// TIA Portal V15.1 export
// export: Created 2024-06-21T08:41:01.5475302Z, ExportSetting WithDefaults, DisplayName Totally Integrated Automation Portal, DisplayVersion V15.1 Update 5, DisplayName TIA Portal Openness, DisplayVersion V15.1 Update 5, DisplayName SINAMICS Startdrive Advanced, DisplayVersion V15.1, DisplayName G130, G150, S120, S150, SINAMICS MV, S210, DisplayVersion V15.1, DisplayName G110M, G120, G120C, G120D, G120P, DisplayVersion V15.1, DisplayName STEP 7 Professional, DisplayVersion V15.1 Update 5, DisplayName STEP 7 Safety, DisplayVersion V15.1, DisplayName WinCC Professional, DisplayVersion V15.1 Update 5, DisplayName SIMATIC Visualization Architect, DisplayVersion V15.1
FUNCTION_BLOCK "LPassivate"   // FB1420, FBD
TITLE = LPassivate
{ S7_Optimized_Access := 'FALSE' }
AUTHOR : VCC
FAMILY : AlarmHnd
NAME : Passivat
VERSION : 0.1
// ================================================================================
// This module is used everywhere passivation of a slot shall generate an alarm.
// The alarm can be True only when the input Enable Alarm is also True.
// When the condition to generate the alarm is not fullfilled, a boolean output is 
// available to inform the upper level that the alarm can be reset.
// The alarm is reset by means of the AlarmResetPB signal.
// ================================================================================
// stored: AutoNumber false, IsIECCheckEnabled false, SetENOAutomatically False, UDAEnableTagReadback false
   VAR_INPUT
      I_SafetyCard_PASS_OUT { ExternalAccessible := 'False'; ExternalVisible := 'False'; ExternalWritable := 'False'} : Bool;   // Automatically generated DB from F-Modul (F-Peripherie DB)
      I_SafetyCard_ACK_REQ { ExternalAccessible := 'False'; ExternalVisible := 'False'; ExternalWritable := 'False'} : Bool;   // Automatically generated DB from F-Modul (F-Peripherie DB)
      I_SafetyCard_DIAG { ExternalAccessible := 'False'; ExternalVisible := 'False'; ExternalWritable := 'False'} : Byte;   // Automatically generated DB from F-Modul (F-Peripherie DB)
      I_SafetyCardHWSub { ExternalAccessible := 'False'; ExternalVisible := 'False'; ExternalWritable := 'False'} : HW_SUBMODULE;   // Safety I/O connection hardware
      I_AlarmClass { ExternalAccessible := 'False'; ExternalVisible := 'False'; ExternalWritable := 'False'} : Char;   // Alarm class -> A - B - C - D or E
      I_EnableAlarm { ExternalAccessible := 'False'; ExternalVisible := 'False'; ExternalWritable := 'False'} : Bool := TRUE;   // Enable alarm from upper level
      I_AlarmResetPB { ExternalAccessible := 'False'; ExternalVisible := 'False'; ExternalWritable := 'False'} : Bool;   // Alarm reset pushbutton is activated
      C_OutputCard { ExternalAccessible := 'False'; ExternalVisible := 'False'; ExternalWritable := 'False'} : Bool;   // 1 = The safety card is an output card
   END_VAR
   VAR_OUTPUT
      O_PassivateAlm { ExternalAccessible := 'False'; ExternalVisible := 'False'; ExternalWritable := 'False'} : Bool;   // Alarm
      O_AlarmABCondition { ExternalAccessible := 'False'; ExternalVisible := 'False'; ExternalWritable := 'False'} : Bool;   // Alarm AB condition
      H_IAnim { ExternalAccessible := 'False'; ExternalVisible := 'False'; ExternalWritable := 'False'} : Word;   // Icon animation
   END_VAR
   VAR DB_SPECIFIC
      H_Out : Struct   // HMI
         Anim : Word;   // HMI Animation of the object
         DBnr : Int;   // HMI Animation DB number
      END_STRUCT;
      Alarm { ExternalAccessible := 'False'; ExternalVisible := 'False'; ExternalWritable := 'False'} : Bool;   // Alarm
      AlarmClass_A { ExternalAccessible := 'False'; ExternalVisible := 'False'; ExternalWritable := 'False'} : Bool;   // The alarm is from alarm class A
      AlarmClass_B { ExternalAccessible := 'False'; ExternalVisible := 'False'; ExternalWritable := 'False'} : Bool;   // The alarm is from alarm class B
      AlarmClass_C { ExternalAccessible := 'False'; ExternalVisible := 'False'; ExternalWritable := 'False'} : Bool;   // The alarm is from alarm class C
      AlarmClass_D { ExternalAccessible := 'False'; ExternalVisible := 'False'; ExternalWritable := 'False'} : Bool;   // The alarm is from alarm class D
      AlarmCond { ExternalAccessible := 'False'; ExternalVisible := 'False'; ExternalWritable := 'False'} : Bool;   // Alarm condition
      QbadCh0 { ExternalAccessible := 'False'; ExternalVisible := 'False'; ExternalWritable := 'False'} : Bool;   // Passivation first Channel
      QbadCh1 { ExternalAccessible := 'False'; ExternalVisible := 'False'; ExternalWritable := 'False'} : Bool;   // Passivation second Channel
      QbadCh2 { ExternalAccessible := 'False'; ExternalVisible := 'False'; ExternalWritable := 'False'} : Bool;   // Passivation third Channel
      QbadCh3 { ExternalAccessible := 'False'; ExternalVisible := 'False'; ExternalWritable := 'False'} : Bool;   // Passivation fourth Channel
      Ack_Req { ExternalAccessible := 'False'; ExternalVisible := 'False'; ExternalWritable := 'False'} : Bool;   // Acknowledgement request
      Pass_Out { ExternalAccessible := 'False'; ExternalVisible := 'False'; ExternalWritable := 'False'} : Bool;   // Slot is passivated
      Timeout_F_I_O { ExternalAccessible := 'False'; ExternalVisible := 'False'; ExternalWritable := 'False'} : Bool;   // Timeout detected by F-I/O
      ChannelFault_F_I_O { ExternalAccessible := 'False'; ExternalVisible := 'False'; ExternalWritable := 'False'} : Bool;   // F-I/O fault or channel fault detected by F-I/O
      CRCSeqError_F_I_O { ExternalAccessible := 'False'; ExternalVisible := 'False'; ExternalWritable := 'False'} : Bool;   // CRC error or sequence number error detected by F-I/O
      Timeout_F_Sys { ExternalAccessible := 'False'; ExternalVisible := 'False'; ExternalWritable := 'False'} : Bool;   // Timeout detected by F-System
      SeqError_F_Sys { ExternalAccessible := 'False'; ExternalVisible := 'False'; ExternalWritable := 'False'} : Bool;   // Sequence number error detected by F-system
      CRCError_F_Sys { ExternalAccessible := 'False'; ExternalVisible := 'False'; ExternalWritable := 'False'} : Bool;   // CRC error detected by F-system
      RetValueData { ExternalAccessible := 'False'; ExternalVisible := 'False'; ExternalWritable := 'False'} : Int;   // Status variable (SFC14)
      DBnr { ExternalAccessible := 'False'; ExternalVisible := 'False'; ExternalWritable := 'False'} : Int;   // HMI DB number
   END_VAR
   VAR_TEMP
      T_DataFromSafetyCard : Struct   // Temp structure : receive data's from Safety Card
         Byte0_Bit0_QBadCh0 : Bool;
         Byte0_Bit1_QBadCh1 : Bool;
         Byte0_Bit2_QBadCh2 : Bool;
         Byte0_Bit3_QBadCh3 : Bool;
         Byte0_Bit4_Spare : Bool;
         Byte0_Bit5_Spare : Bool;
         Byte0_Bit6_Spare : Bool;
         Byte0_Bit7_Spare : Bool;
         Byte1_Bit0_QBadCh0 : Bool;
         Byte1_Bit1_QBadCh1 : Bool;
         Byte1_Bit2_QBadCh2 : Bool;
         Byte1_Bit3_QBadCh3 : Bool;
         Byte1_Bit4_Spare : Bool;
         Byte1_Bit5_Spare : Bool;
         Byte1_Bit6_Spare : Bool;
         Byte1_Bit7_Spare : Bool;
         Byte2_bit0_Spare : Bool;
         Byte2_bit1_Spare : Bool;
         Byte2_bit2_Spare : Bool;
         Byte2_bit3_Spare : Bool;
         Byte2_bit4_Spare : Bool;
         Byte2_bit5_Spare : Bool;
         Byte2_bit6_Spare : Bool;
         Byte2_bit7_Spare : Bool;
         Byte3_Bit0_Spare : Bool;
         Byte3_Bit1_Spare : Bool;
         Byte3_Bit2_Spare : Bool;
         Byte3_Bit3_Spare : Bool;
         Byte3_Bit4_Spare : Bool;
         Byte3_Bit5_Spare : Bool;
         Byte3_Bit6_Spare : Bool;
         Byte3_Bit7_Spare : Bool;
         Byte4_bit0_Spare : Bool;
         Byte4_bit1_Spare : Bool;
         Byte4_bit2_Spare : Bool;
         Byte4_bit3_Spare : Bool;
         Byte4_bit4_Spare : Bool;
         Byte4_bit5_Spare : Bool;
         Byte4_bit6_Spare : Bool;
         Byte4_bit7_Spare : Bool;
         Byte5_bit0_Spare : Bool;
         Byte5_bit1_Spare : Bool;
         Byte5_bit2_Spare : Bool;
         Byte5_bit3_Spare : Bool;
         Byte5_bit4_Spare : Bool;
         Byte5_bit5_Spare : Bool;
         Byte5_bit6_Spare : Bool;
         Byte5_bit7_Spare : Bool;
      END_STRUCT;
   END_VAR
BEGIN

NETWORK
TITLE = **** 1 - Inputs **** DB number
// DB number
      L     DINO;
      T     #DBnr;

NETWORK
TITLE = **** 1 - Inputs **** Alarm class
// Alarm class
// Alarm class = D
      L     #I_AlarmClass;
      L     'D';
      ==I;
      =     #AlarmClass_D;

// Alarm class = C
      L     #I_AlarmClass;
      L     'C';
      ==I;
      =     #AlarmClass_C;

// Alarm class = B
      L     #I_AlarmClass;
      L     'B';
      ==I;
      =     #AlarmClass_B;

// Alarm class = A
      AN    #AlarmClass_B;
      AN    #AlarmClass_C;
      AN    #AlarmClass_D;
      =     #AlarmClass_A;


REGION Network 3: **** 1 - Inputs **** Safety I/O connection hardware
   // Safety I/O connection hardware
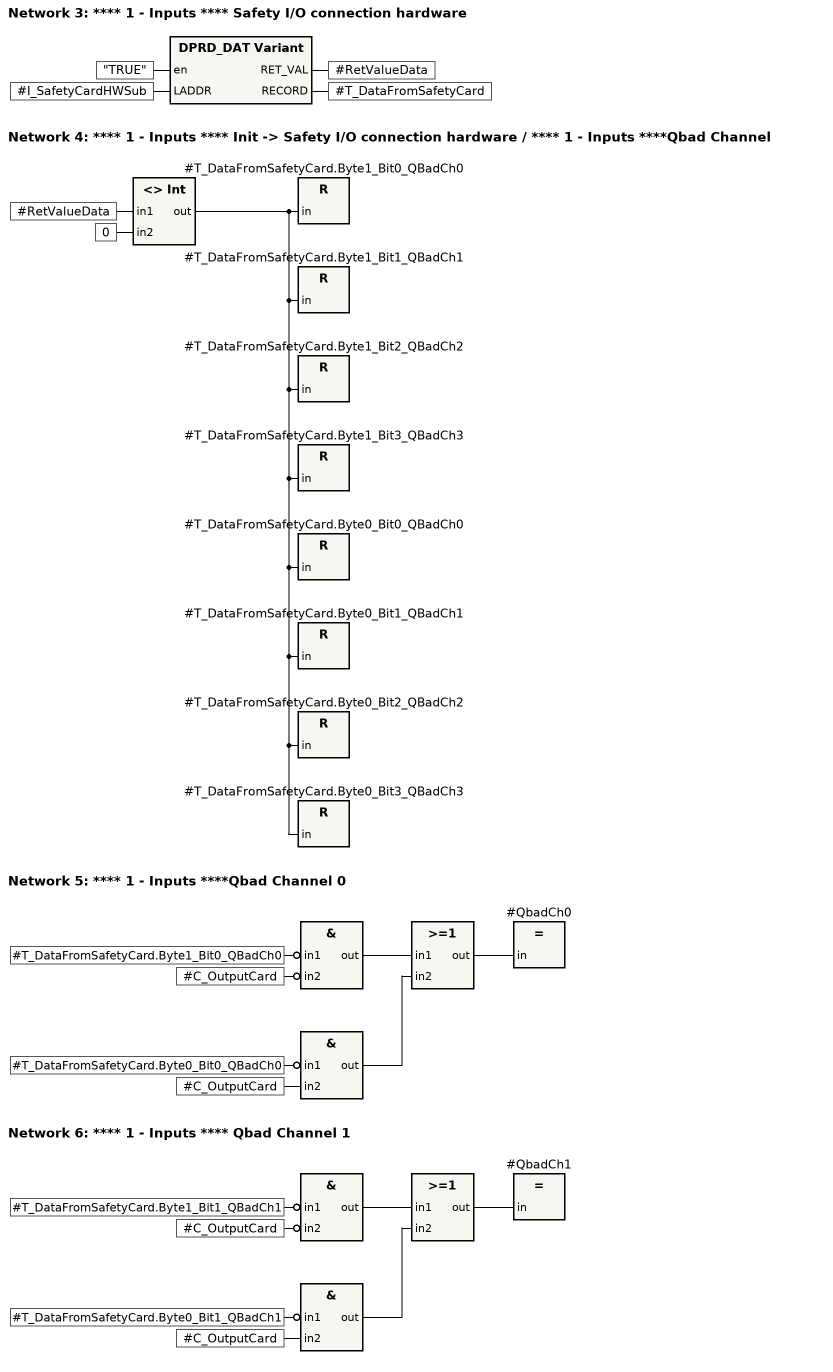
   IF "TRUE" THEN
       #RetValueData := DPRD_DAT(LADDR := #I_SafetyCardHWSub, RECORD => #T_DataFromSafetyCard);
   END_IF;
END_REGION

REGION Network 4: **** 1 - Inputs **** Init -> Safety I/O connection hardware / **** 1 - Inputs ****Qbad Channel
   // Init -> Safety I/O connection hardware
   IF #RetValueData <> 0 THEN
       #T_DataFromSafetyCard.Byte1_Bit0_QBadCh0 := FALSE;
       #T_DataFromSafetyCard.Byte1_Bit1_QBadCh1 := FALSE;
       #T_DataFromSafetyCard.Byte1_Bit2_QBadCh2 := FALSE;
       #T_DataFromSafetyCard.Byte1_Bit3_QBadCh3 := FALSE;
       #T_DataFromSafetyCard.Byte0_Bit0_QBadCh0 := FALSE;
       #T_DataFromSafetyCard.Byte0_Bit1_QBadCh1 := FALSE;
       #T_DataFromSafetyCard.Byte0_Bit2_QBadCh2 := FALSE;
       #T_DataFromSafetyCard.Byte0_Bit3_QBadCh3 := FALSE;
   END_IF;
END_REGION

REGION Network 5: **** 1 - Inputs ****Qbad Channel 0
   // Qbad Channel 0
   #QbadCh0 := (NOT #T_DataFromSafetyCard.Byte1_Bit0_QBadCh0 AND NOT #C_OutputCard) OR (NOT #T_DataFromSafetyCard.Byte0_Bit0_QBadCh0 AND #C_OutputCard);
END_REGION

REGION Network 6: **** 1 - Inputs **** Qbad Channel 1
   // Qbad Channel 1
   #QbadCh1 := (NOT #T_DataFromSafetyCard.Byte1_Bit1_QBadCh1 AND NOT #C_OutputCard) OR (NOT #T_DataFromSafetyCard.Byte0_Bit1_QBadCh1 AND #C_OutputCard);
END_REGION

REGION Network 7: **** 1 - Inputs **** Qbad Channel 2
   // Qbad Channel 2
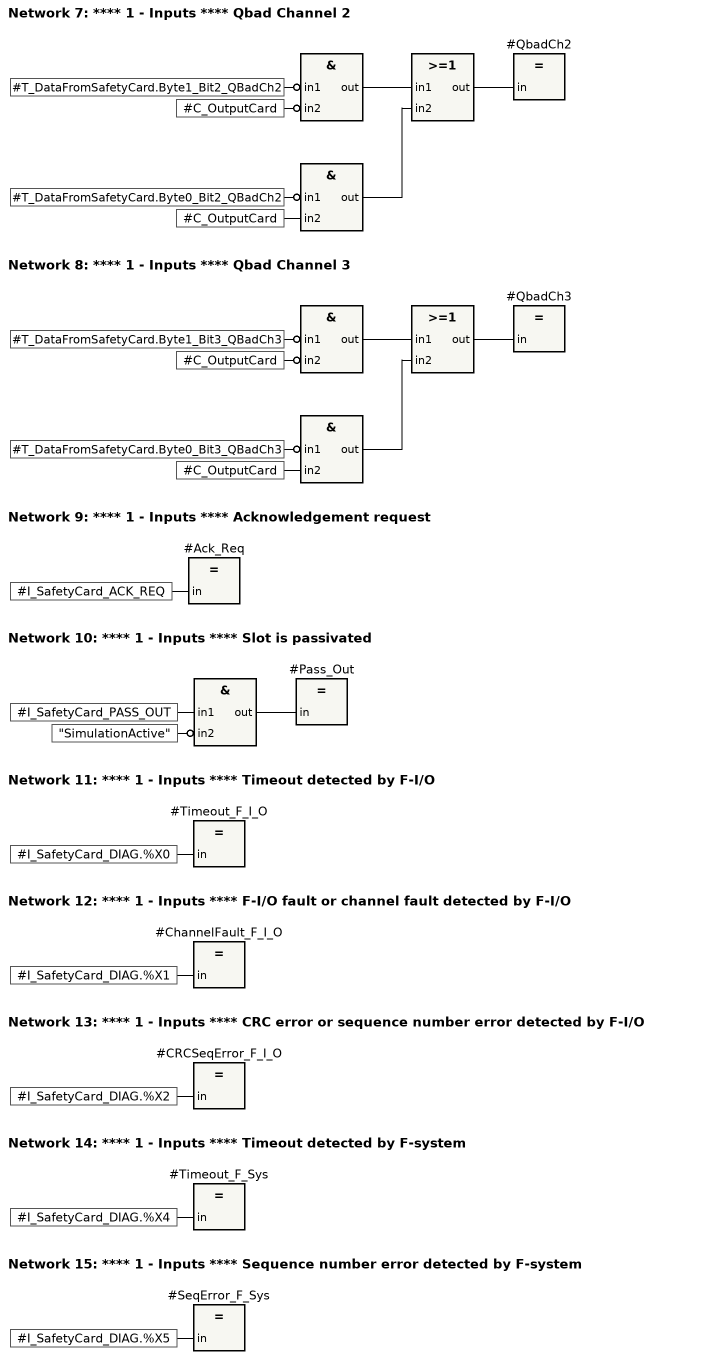
   #QbadCh2 := (NOT #T_DataFromSafetyCard.Byte1_Bit2_QBadCh2 AND NOT #C_OutputCard) OR (NOT #T_DataFromSafetyCard.Byte0_Bit2_QBadCh2 AND #C_OutputCard);
END_REGION

REGION Network 8: **** 1 - Inputs **** Qbad Channel 3
   // Qbad Channel 3
   #QbadCh3 := (NOT #T_DataFromSafetyCard.Byte1_Bit3_QBadCh3 AND NOT #C_OutputCard) OR (NOT #T_DataFromSafetyCard.Byte0_Bit3_QBadCh3 AND #C_OutputCard);
END_REGION

REGION Network 9: **** 1 - Inputs **** Acknowledgement request
   // Acknowledgement request
   #Ack_Req := #I_SafetyCard_ACK_REQ;
END_REGION

REGION Network 10: **** 1 - Inputs **** Slot is passivated
   // Slot is passivated
   #Pass_Out := #I_SafetyCard_PASS_OUT AND NOT "SimulationActive";
END_REGION

REGION Network 11: **** 1 - Inputs **** Timeout detected by F-I/O
   // Timeout detected by F-I/O
   #Timeout_F_I_O := #I_SafetyCard_DIAG.%X0;
END_REGION

REGION Network 12: **** 1 - Inputs **** F-I/O fault or channel fault detected by F-I/O
   // F-I/O fault or channel fault detected by F-I/O
   #ChannelFault_F_I_O := #I_SafetyCard_DIAG.%X1;
END_REGION

REGION Network 13: **** 1 - Inputs **** CRC error or sequence number error detected by F-I/O
   // CRC error or sequence number error detected by F-I/O
   #CRCSeqError_F_I_O := #I_SafetyCard_DIAG.%X2;
END_REGION

REGION Network 14: **** 1 - Inputs **** Timeout detected by F-system
   // Timeout detected by F-system
   #Timeout_F_Sys := #I_SafetyCard_DIAG.%X4;
END_REGION

REGION Network 15: **** 1 - Inputs **** Sequence number error detected by F-system
   // Sequence number error detected by F-system
   #SeqError_F_Sys := #I_SafetyCard_DIAG.%X5;
END_REGION

REGION Network 16: **** 1 - Inputs **** CRC error detected by F-system
   // CRC error detected by F-system
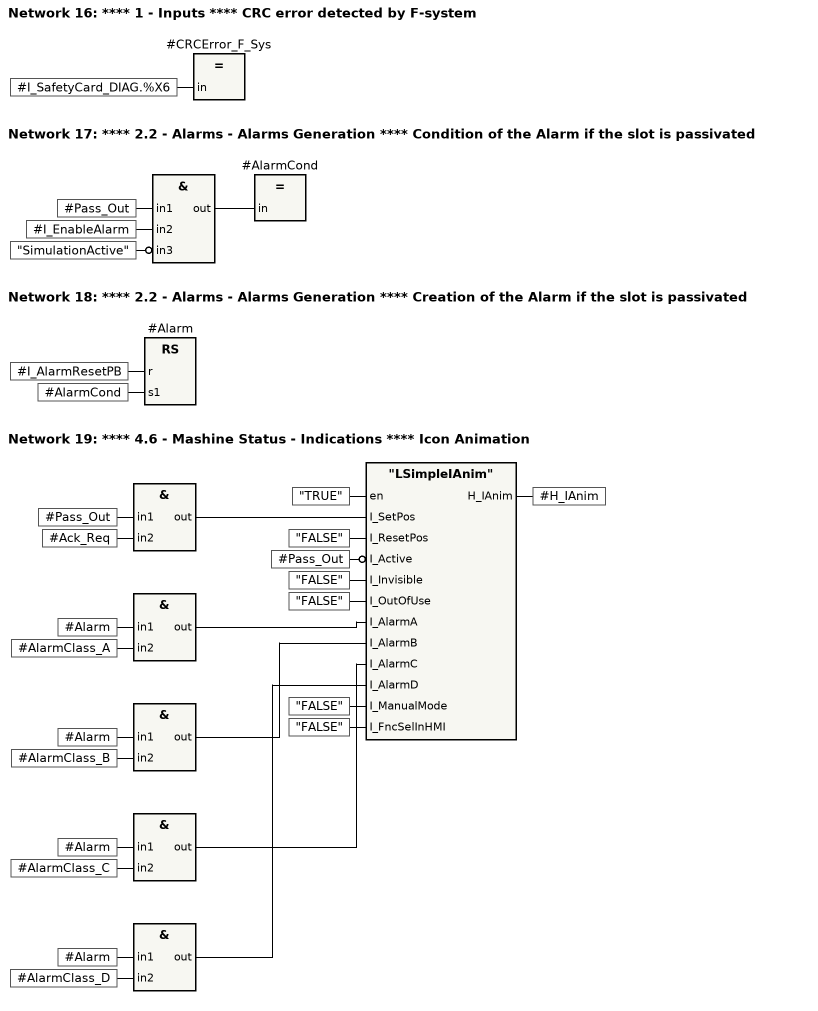
   #CRCError_F_Sys := #I_SafetyCard_DIAG.%X6;
END_REGION

REGION Network 17: **** 2.2 - Alarms - Alarms Generation **** Condition of the Alarm if the slot is passivated
   // Condition of the Alarm if the slot is passivated
   #AlarmCond := #Pass_Out AND #I_EnableAlarm AND NOT "SimulationActive";
END_REGION

REGION Network 18: **** 2.2 - Alarms - Alarms Generation **** Creation of the Alarm if the slot is passivated
   // Creation of the Alarm if the slot is passivated
   IF #I_AlarmResetPB THEN
       #Alarm := FALSE;   // RS flip-flop
   END_IF;
   IF #AlarmCond THEN #Alarm := TRUE; END_IF;
END_REGION

REGION Network 19: **** 4.6 - Mashine Status - Indications **** Icon Animation
   // Icon Animation
   IF "TRUE" THEN
       "LSimpleIAnim"(I_SetPos := #Pass_Out AND #Ack_Req,
                      I_ResetPos := "FALSE",
                      I_Active := NOT #Pass_Out,
                      I_Invisible := "FALSE",
                      I_OutOfUse := "FALSE",
                      I_AlarmA := #Alarm AND #AlarmClass_A,
                      I_AlarmB := #Alarm AND #AlarmClass_B,
                      I_AlarmC := #Alarm AND #AlarmClass_C,
                      I_AlarmD := #Alarm AND #AlarmClass_D,
                      I_ManualMode := "FALSE",
                      I_FncSelInHMI := "FALSE",
                      H_IAnim => #H_IAnim);
   END_IF;
END_REGION

REGION Network 20: **** 4.6 - Mashine Status - Indications **** Animation
   // Animation
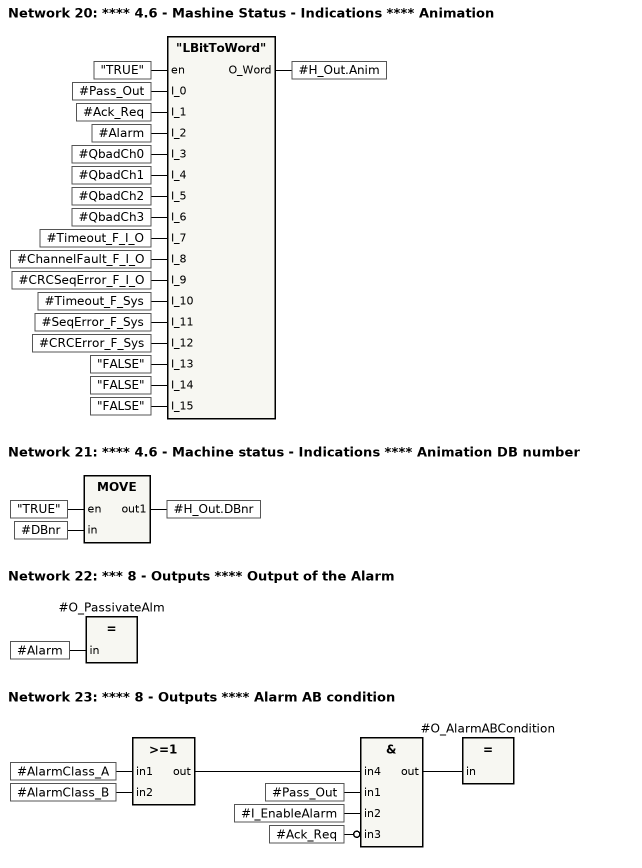
   IF "TRUE" THEN
       "LBitToWord"(I_0 := #Pass_Out,
                    I_1 := #Ack_Req,
                    I_2 := #Alarm,
                    I_3 := #QbadCh0,
                    I_4 := #QbadCh1,
                    I_5 := #QbadCh2,
                    I_6 := #QbadCh3,
                    I_7 := #Timeout_F_I_O,
                    I_8 := #ChannelFault_F_I_O,
                    I_9 := #CRCSeqError_F_I_O,
                    I_10 := #Timeout_F_Sys,
                    I_11 := #SeqError_F_Sys,
                    I_12 := #CRCError_F_Sys,
                    I_13 := "FALSE",
                    I_14 := "FALSE",
                    I_15 := "FALSE",
                    O_Word => #H_Out.Anim);
   END_IF;
END_REGION

REGION Network 21: **** 4.6 - Machine status - Indications **** Animation DB number
   // Animation DB number
   IF "TRUE" THEN #H_Out.DBnr := #DBnr; END_IF;
END_REGION

REGION Network 22: *** 8 - Outputs **** Output of the Alarm
   // Output of the Alarm
   #O_PassivateAlm := #Alarm;
END_REGION

REGION Network 23: **** 8 - Outputs **** Alarm AB condition
   // Alarm AB condition
   #O_AlarmABCondition := (#AlarmClass_A OR #AlarmClass_B) AND #Pass_Out AND #I_EnableAlarm AND NOT #Ack_Req;
END_REGION
END_FUNCTION_BLOCK
